{attribute 'qualified_only'}
{attribute 'strict'}
TYPE ButtonStatus :
(
	UNKNOWN := 0, 
	RELEASED := 1, 
	PRESSED := 2
);
END_TYPE

(* stored: Version 1.1.0.1, ProductVersion 3.1.4024.12
   DUT ButtonStatus: Id {09185448-9596-44d4-b71e-9a8730f6048d} *)
